Fanuc KAREL source: compact_preamble.KL

PROGRAM KT00894
%NOLOCKGROUP
VAR
P1 : XYZWPR;P2 : XYZWPR;OUT:BOOLEAN
BEGIN
P1.X=1.0
P2.Y=2.0
P1.X=1.0
P2.Y=2.0
OUT=IN_RANGE(P1)
END KT00894
